# B&R Automation Studio project Task_2
Automation Studio 4.9

## Logical view

Binary libraries used (declarations not repeated): operator, runtime, astime, AsIecCon, Acp10man, Acp10par, NcGlobal, Acp10_MC, sys_lib, brsystem, Acp10sim, MpAxis, MpCom, MpBase, AsTCP, standard, AsArLog, AsBrStr

### Global.var - Global variables
```iecst
VAR
	EmergencyLight : BOOL;
END_VAR
VAR RETAIN
	MyGlobal : {REDUND_UNREPLICABLE} UDINT := 10;
END_VAR
VAR
	CUTTER_END_POSE : REAL := 50.0;
END_VAR
VAR CONSTANT
	BELT_DISTANCE : REAL := 100.0;
	CUTTER_SPEED : REAL := 100.0;
END_VAR
VAR
	RealConveyorSpeed : INT;
	CONVEYOR_SPEED : {REDUND_UNREPLICABLE} INT := 1000;
	gAxis01 : ACP10AXIS_typ;
	gAxis02 : ACP10AXIS_typ;
	START_BUTTON : BOOL;
	TRIGGER_INPUT : BOOL;
	EMERGENCY_STOP : BOOL;
	GreenLight : BOOL;
	RedLight : BOOL;
	CutterPosition : LREAL;
	ConveyorPosition : LREAL;
	STOP : BOOL;
	ERROR_RESET : BOOL;
END_VAR
```

### Package Logical/Libraries - Global libraries

### MNG_Global.hpp
```cpp
#ifndef  _MNGGLOBAL_HPP_
#define _MNGGLOBAL_HPP_

#include <mng_globalTYP.h>

    typedef struct {

		signed short NumSignals;

        /* BOOL Emergency_Button_ButtonToggle */
        BOOL Emergency_Button_ButtonToggle;
        /* BOOL Yellow_Button_ButtonPress */
        BOOL Yellow_Button_ButtonPress;
        /* BOOL White_Button_ButtonPress */
        BOOL White_Button_ButtonPress;
        /* BOOL Start_Button_ButtonPress */
        BOOL Start_Button_ButtonPress;
        /* BOOL Stop_Button_ButtonPress */
        BOOL Stop_Button_ButtonPress;
        /* REAL Knob_0_AXIS */
        REAL Knob_0_AXIS;
        /* REAL Knob_1_AXIS */
        REAL Knob_1_AXIS;
        /* REAL Knob_2_AXIS */
        REAL Knob_2_AXIS;
        /* REAL Knob_3_AXIS */
        REAL Knob_3_AXIS;
        /* REAL Shaft_1_AXIS */
        REAL Shaft_1_AXIS;
        /* BOOL Shaft_1_LBK */
        BOOL Shaft_1_LBK;
        /* BOOL Shaft_1_LFR */
        BOOL Shaft_1_LFR;
        /* REAL Shaft_0_AXIS */
        REAL Shaft_0_AXIS;
        /* BOOL Shaft_0_LBK */
        BOOL Shaft_0_LBK;
        /* BOOL Shaft_0_LFR */
        BOOL Shaft_0_LFR;

        } ComTCP_INPUTS_32BIT_FWRD;

    typedef struct {

		signed short NumSignals;

        /* UDINT Yellow_light_Key */
        UDINT Yellow_light_Key;
        /* UDINT Stop_light_Key */
        UDINT Stop_light_Key;
        /* UDINT White_light_Key */
        UDINT White_light_Key;
        /* UDINT Green_light_Key */
        UDINT Green_light_Key;
        /* REAL Shaft_0_ACT_POS */
        REAL Shaft_0_ACT_POS;
        /* REAL Shaft_1_ACT_POS */
        REAL Shaft_1_ACT_POS;

        } ComTCP_OUTPUTS_32BIT_FWRD;

#endif
```

### Library Logical/Libraries/CAMlib (IEC)

#### Types.typ - Exported data types
```iecst
TYPE
	GA_State :
		(
		NotPowered,
		WaitEnable,
		WaitPower,
		Powered,
		CheckCommand,
		MoveVelocity,
		CheckVelocity,
		MoveAdditive,
		CheckAdditiveUpdate,
		AxisHalt,
		AxisStop,
		CheckCamUpdate,
		CheckCam,
		MoveCam,
		CheckVelocityUpdate,
		AxisEmergency
		);
	COMMANDS :
		(
		NONE,
		MOVE_VELOCITY,
		MOVE_ADDITIVE,
		AXIS_HALT,
		AXIS_STOP,
		MOVE_CAM,
		AXIS_EMERGENCY
		);
END_TYPE
```

#### CAMlib.fun - Exported functions and function blocks
```iecst
{REDUND_ERROR} FUNCTION_BLOCK CamFB (*TODO: Add your comment here*) (*$GROUP=User,$CAT=User,$GROUPICON=User.png,$CATICON=User.png*)
	VAR_INPUT
		AxisOperation : INT;
		AxisCommand : COMMANDS;
		Axis : UDINT;
		MpLinkMaster : UDINT;
		MpLink : UDINT;
		Slave : UDINT;
		CamTable : ARRAY[0..4] OF STRING[12];
		Position : REAL;
		Velocity : REAL;
		Acceleration : REAL;
		Deceleration : REAL;
		Jerk : REAL;
		Direction : USINT;
		ArraySize : INT;
		Scale : REAL;
		Offset : REAL;
		RatioNumerator : INT;
		CamID : USINT;
		CamActivated : BOOL;
		RatioDenominator : INT;
		CouplingParam : MpAxisCouplingParType;
		Param : MpAxisBasicParType;
	END_VAR
	VAR_OUTPUT
		CommandExecuted : BOOL;
		CommandAborted : BOOL;
		Error : BOOL;
		ErrorID : UINT;
		AxisErrorID : UINT;
		AxisErrorCount : UINT;
		AxisNotInitialized : BOOL;
		Status : WORD;
		ActualVelocity : REAL;
		ActualPosition : LREAL;
	END_VAR
	VAR_IN_OUT
		AxisEnable : BOOL;
	END_VAR
	VAR
		MpAxisCoupling : MpAxisCoupling;
		MpAxisBasic : MpAxisBasic;
		OldVelocity : REAL;
		AxisState : GA_State;
		OldCamID : USINT;
	END_VAR
END_FUNCTION_BLOCK
```

#### CamFB.st
```iecst
(* TODO: Add your comment here *)
FUNCTION_BLOCK CamFB

	CASE (AxisState) OF
		NotPowered:
			IF AxisEnable THEN
				MpAxisBasic.Enable := TRUE;
				AxisState := WaitEnable;
			END_IF;

		WaitEnable:
			IF MpAxisBasic.Active THEN
				MpAxisBasic.Power := TRUE;
				AxisState := WaitPower; //ready state in the prof's slides
			END_IF;

		WaitPower:
			IF  MpAxisBasic.PowerOn THEN
				MpAxisBasic.Home := TRUE;
				AxisState := Powered;
			END_IF;

		Powered:
			IF MpAxisBasic.IsHomed THEN // condition for the homing
				MpAxisBasic.Home := FALSE;
				AxisEnable := FALSE;
				CommandExecuted := TRUE;
				MpAxisCoupling.Enable := TRUE;
				AxisState := CheckCommand; //ready state in the prof's slides
			END_IF;

		CheckCommand:
			IF AxisCommand = MOVE_VELOCITY THEN
				CommandExecuted := FALSE;
				MpAxisBasic.MoveAdditive := FALSE;
				MpAxisBasic.Update := TRUE;
				// MpAxisBasic.MoveVelocity := TRUE;  // <------ Come se ricevesse velocità nulla
				AxisState := CheckVelocityUpdate;
			END_IF;

			IF AxisCommand = MOVE_ADDITIVE THEN
				CommandExecuted := FALSE;
				MpAxisBasic.MoveVelocity := FALSE;
				MpAxisBasic.MoveAdditive := TRUE;
				MpAxisBasic.Update := TRUE;
				AxisState := CheckAdditiveUpdate; //CheckAdditiveUpdate;
			END_IF;

			IF AxisCommand = AXIS_STOP THEN
				CommandExecuted := FALSE;
				MpAxisBasic.MoveVelocity := FALSE;
				MpAxisBasic.MoveAdditive := FALSE;
				MpAxisBasic.Stop := TRUE;
				AxisState := AxisStop;
			END_IF;

			IF AxisCommand = AXIS_EMERGENCY THEN
				CommandExecuted := FALSE;
				MpAxisBasic.MoveVelocity := FALSE;
				MpAxisBasic.MoveAdditive := FALSE;
				MpAxisBasic.Stop := TRUE;
				AxisState := AxisEmergency;
			END_IF;

			IF AxisCommand = MOVE_CAM AND CamActivated THEN
				CommandExecuted := FALSE;
				MpAxisCoupling.Cam := TRUE;
				AxisState := MoveCam;
			END_IF;

	(*IF AxisCommand = NONE THEN
		CommandExecuted := FALSE;
	END_IF*)

// command states
		MoveVelocity:
			IF MpAxisBasic.InVelocity THEN  // <------- Siccome la velocità è nulls lo esegue subito
				CommandExecuted := TRUE;
				AxisState := CheckVelocity;
			END_IF;

			IF (AxisCommand <> MOVE_VELOCITY) THEN
				CommandExecuted := FALSE;
				MpAxisBasic.MoveVelocity := FALSE;
				AxisState := CheckCommand;
			END_IF;

		CheckVelocity:
			IF (Param.Velocity <> OldVelocity) THEN
				OldVelocity := Param.Velocity;
				MpAxisBasic.Update := TRUE;
				AxisState := CheckVelocityUpdate;
			END_IF;
			IF (AxisCommand <> MOVE_VELOCITY) THEN
				CommandExecuted := FALSE;
				MpAxisBasic.MoveVelocity := FALSE;
				AxisState := CheckCommand;
			END_IF;

		CheckVelocityUpdate:
			IF MpAxisBasic.UpdateDone THEN
				MpAxisBasic.Update := FALSE;
				MpAxisBasic.MoveVelocity := TRUE;
				CommandExecuted := FALSE;
				AxisState := MoveVelocity;
			END_IF;

		MoveAdditive:
			IF MpAxisBasic.InPosition THEN
				MpAxisBasic.MoveAdditive := FALSE;
				AxisCommand := NONE;
				AxisState := CheckCommand;
				CommandExecuted := TRUE;
			ELSIF (AxisCommand <> MOVE_ADDITIVE) THEN
				MpAxisBasic.MoveAdditive := FALSE;
				CommandExecuted := FALSE;
				AxisState := CheckCommand;
			END_IF;

		CheckAdditiveUpdate:
			IF MpAxisBasic.UpdateDone THEN
				MpAxisBasic.Update := FALSE;
				MpAxisBasic.MoveAdditive := TRUE;
				CommandExecuted := FALSE;
					AxisState := MoveAdditive;
			END_IF;

		AxisStop:
			IF MpAxisBasic.Stopped THEN
				CommandExecuted := TRUE;
				MpAxisBasic.Stop := FALSE;
				MpAxisBasic.Power := FALSE; // The power is disabled for the same reason
				// MpAxisBasic.Enable := FALSE;
				// MpAxisCoupling.Enable := FALSE;
				MpAxisCoupling.Cam := FALSE;
				AxisCommand := NONE;
				AxisState := NotPowered; // It goes to the NotPowered state to perform a full reset of the system
			END_IF;

		AxisEmergency:
			IF MpAxisBasic.Stopped THEN
				CommandExecuted := TRUE;
				MpAxisBasic.Stop := FALSE;
				MpAxisBasic.Power := FALSE; // The power is disabled for the same reason
				// MpAxisBasic.Enable := FALSE;
				// MpAxisCoupling.Enable := FALSE;
				MpAxisCoupling.Cam := FALSE;
				AxisCommand := NONE;
				AxisState := NotPowered; // It goes to the NotPowered state to perform a full reset of the system
			END_IF;

			// memo, we don't check the mpaxiscoupling.active -> WARNING

		MoveCam:
			IF MpAxisCoupling.InSync THEN
				CommandExecuted := TRUE;
				AxisState := CheckCam;
			END_IF
			IF (AxisCommand <> MOVE_CAM) THEN
				CommandExecuted := FALSE;
				MpAxisCoupling.Cam := FALSE;
				MpAxisCoupling.Enable := FALSE;
				AxisState := CheckCommand;
			END_IF;
		CheckCam:
			IF CamID <> OldCamID THEN
				OldCamID := CamID;
				CommandExecuted := FALSE;
				MpAxisCoupling.Update := TRUE;
				AxisState := CheckCamUpdate;
			END_IF
			IF (AxisCommand <> MOVE_CAM) THEN
				CommandExecuted := FALSE;
				MpAxisCoupling.Cam := FALSE;
				MpAxisCoupling.Enable := FALSE;
				AxisState := CheckCommand;
			END_IF;

		CheckCamUpdate:
			IF MpAxisCoupling.UpdateDone THEN
				MpAxisCoupling.Update := FALSE;
				AxisState := MoveCam;
			END_IF;

	END_CASE

	MpAxisBasic.Axis := Axis;
	MpAxisBasic.MpLink := MpLink;

	MpAxisBasic.Parameters	:= ADR(Param);
	ActualPosition := MpAxisBasic.Position;

	MpAxisBasic();

	IF CamActivated THEN
		MpAxisCoupling.MpLinkMaster	:= MpLinkMaster;
		MpAxisCoupling.MpLink := MpLink;
		CouplingParam.Cam.CamTableID := CamID;
		CouplingParam.Cam.CamTable := CamTable;
		MpAxisCoupling.Parameters := ADR(CouplingParam);
		MpAxisCoupling();
	END_IF

END_FUNCTION_BLOCK
```

### Package Logical/gAxis02obj - gAxis02obj

### gAxis02i.ax
```
InitParameter (Version=5.24.1, NcSwId=Acp10)
  ACP10AXIS_typ:
    dig_in:
      level:
        reference = ncACTIV_HI
        pos_hw_end = ncACTIV_HI
        neg_hw_end = ncACTIV_HI
        trigger1 = ncACTIV_HI
        trigger2 = ncACTIV_HI
    encoder_if:
      parameter:
        count_dir = ncSTANDARD
        scaling:
          load:
            units = 360
            rev_motor = 1
    limit:
      parameter:
        v_pos = 10000
        v_neg = 10000
        a1_pos = 50000
        a2_pos = 50000
        a1_neg = 50000
        a2_neg = 50000
        t_jolt = 0
        t_in_pos = 0
        pos_sw_end = 2000000000
        neg_sw_end = -2000000000
        ds_warning = 500
        ds_stop = 1000
        a_stop = 1.0e30
        dv_stop = 0
        dv_stop_mode = ncOFF
    controller:
      mode = ncPOSITION
      position:
        kv = 349.0
        tn = 0
        t_predict = 0.0004
        t_total = 0.0004
        p_max = 1.0e30
        i_max = 0
      speed:
        kv = 0.65
        tn = 0
        t_filter = 0.0
        isq_filter1:
          type = ncOFF
          a0 = 0.0
          a1 = 0.0
          b0 = 0.0
          b1 = 0.0
          b2 = 0.0
          c0_par_id = 0
          c1_par_id = 0
        isq_filter2:
          type = ncOFF
          a0 = 0.0
          a1 = 0.0
          b0 = 0.0
          b1 = 0.0
          b2 = 0.0
          c0_par_id = 0
          c1_par_id = 0
        isq_filter3:
          type = ncOFF
          a0 = 0.0
          a1 = 0.0
          b0 = 0.0
          b1 = 0.0
          b2 = 0.0
          c0_par_id = 0
          c1_par_id = 0
      uf:
        type = ncLINEAR + ncCORRECTION
        auto_config = ncMOTOR_PAR
        u0 = 0
        un = 0
        fn = 50.0
        k_f_slip = 0
      ff:
        mode = ncSTANDARD
        torque_load = 0.0
        torque_pos = 0.0
        torque_neg = 0.0
        kv_torque = 0.0
        inertia = 0.0
        t_filter_a = 0.0
      fb:
        mode = ncSTANDARD
        speed_mix_ratio = 0.0
        speed_kv = 2.0
      model:
        mass1:
          inertia = 0
          viscous_friction = 0
        mass2:
          inertia = 0
          viscous_friction = 0
          stiffness = 0
          damping = 0
    move:
      stop:
        parameter[0]:
          decel_ramp = ncA_LIMIT
          controller = ncON
        parameter[1]:
          decel_ramp = ncA_LIMIT
          controller = ncON
        parameter[2]:
          decel_ramp = ncA_LIMIT
          controller = ncON
        parameter[3]:
          decel_ramp = ncA_LIMIT
          controller = ncON
        quickstop:
          decel_ramp = ncA_LIMIT
          t_jolt = 0
        drive_error:
          decel_ramp = ncA_LIMIT
      homing:
        parameter:
          s = 0
          v_switch = 5000
          v_trigger = 500
          a = 50000
          mode = ncDIRECT
          edge_sw = ncPOSITIVE
          start_dir = ncPOSITIVE
          trigg_dir = ncPOSITIVE
          ref_pulse = ncOFF
          fix_dir = ncOFF
          tr_s_block = 0
          torque_lim = 0
          ds_block = 0
          ds_stop = 0
      basis:
        parameter:
          v_pos = 5000
          v_neg = 5000
          a1_pos = 50000
          a2_pos = 50000
          a1_neg = 50000
          a2_neg = 50000
    message:
      text:
        parameter:
          format = ncBREAK
          columns = 80
          data_modul = acp10etxen
```

### Program Logical/PROGRAM1 (IEC)

#### Types.typ
```iecst
TYPE
	State_type :
		(
		CutterMoveBackward,
		CutterCompleted,
		CutterMoveForward,
		ConveyorStopping,
		ConveyorMoving,
		ConveyorStarting,
		AxisEnabled,
		InitializeAxis,
		CutterBackward,
		CutterForward,
		ConveyorHolding,
		WaitProduct,
		Initialize,
		Init,
		StopState,
		HaltState,
		WaitForConveyor,
		CheckReset
		);
END_TYPE
```

#### Variables.var
```iecst
VAR
	Address : UDINT;
	MachineState : State_type;
	ConveyorEnable : BOOL;
	CutterEnable : BOOL;
	Cutter : CamFB;
	Conveyor : CamFB;
	InitializeConveyor : BOOL;
	InitializeCutter : BOOL;
	ConveyorDisable : BOOL;
	CutterDisable : BOOL;
	ConveyorState : State_type;
	CutterState : State_type;
	ConveyorAxisEnable : BOOL;
	CutterAxisEnable : BOOL;
	FutureStop : BOOL;
	CoveyorState : BOOL;
	ConveyorStopped : BOOL;
	CutterStopped : BOOL;
	ConveyorParameters : MpAxisBasicParType;
	CutterParameters : MpAxisBasicParType;
	EmergencyStateMachine : INT;
	ToggleLights : BOOL;
	Count : DINT;
END_VAR
```

#### Main.st
```iecst
PROGRAM _INIT
	(* Insert code here *)
	MachineState := Init;
	ConveyorState := Init;
	CutterState := Init;

END_PROGRAM

PROGRAM _CYCLIC

	// STOP indicates an emergency stop, it is not a stop in normal conditions
	CASE EmergencyStateMachine OF
		0 :
			IF EMERGENCY_STOP THEN
				MachineState := StopState;
				ConveyorState := StopState;
				CutterState := StopState;
				Conveyor.AxisCommand := AXIS_STOP;
				Cutter.AxisCommand := AXIS_STOP;
				EmergencyStateMachine := 1;
			END_IF
		1 :
			IF NOT EMERGENCY_STOP AND CutterStopped AND ConveyorStopped THEN
				EmergencyStateMachine := 0;
			END_IF
	END_CASE

	IF STOP THEN
		FutureStop := TRUE;
	END_IF

	// GLOBAL STATE MACHINE
	CASE MachineState OF
		Init: // Initial configuration state
			IF START_BUTTON THEN
				InitializeConveyor := TRUE;
				InitializeCutter := TRUE;
				MachineState := Initialize;
			END_IF
		Initialize: // initialization - Power and Homing (This operations are implemented inside the function block)
			IF NOT InitializeConveyor AND NOT InitializeCutter THEN
				ConveyorEnable := TRUE;
				MachineState := WaitProduct;
			END_IF
		WaitProduct: // It waits for a trigger
			IF NOT ConveyorEnable AND TRIGGER_INPUT THEN
				ConveyorDisable := TRUE;
				MachineState := ConveyorHolding;
			END_IF
			// STOP
			IF FutureStop THEN
				MachineState := HaltState;
			END_IF

		ConveyorHolding: // Stop the Conveyor
			IF NOT ConveyorDisable THEN
				CutterEnable := TRUE;
				MachineState := CutterForward;
			END_IF
		CutterForward: // Cut
			IF NOT CutterEnable THEN
				CutterDisable := TRUE;
				MachineState := CutterBackward;
			END_IF
		CutterBackward: // Go back
			IF NOT CutterDisable THEN
				ConveyorEnable := TRUE;
				MachineState := WaitProduct;
			END_IF

		// Emergency stop
		StopState:
			IF NOT EMERGENCY_STOP AND ConveyorStopped AND CutterStopped THEN
				MachineState := CheckReset;
			END_IF
		CheckReset:
			IF ERROR_RESET THEN
				MachineState := Init;
				ConveyorStopped := FALSE;
				CutterStopped := FALSE;
				FutureStop := FALSE;
			END_IF
			// CAN BE ERASED
		// CAN BE ERASED
		HaltState:
			IF ConveyorStopped AND CutterStopped THEN
				MachineState := Init;
				ConveyorStopped := FALSE;
				CutterStopped := FALSE;
				FutureStop := FALSE;
			END_IF

	END_CASE

	// CONVEYOR STATE MACHINE
	CASE ConveyorState OF
		Init:
			IF InitializeConveyor THEN
				ConveyorAxisEnable := TRUE;
				ConveyorState := InitializeAxis;
			END_IF
		InitializeAxis:
			IF NOT ConveyorAxisEnable THEN
				InitializeConveyor := FALSE;
				ConveyorState := AxisEnabled;
			END_IF
		AxisEnabled:
			IF ConveyorEnable AND NOT FutureStop THEN
				Conveyor.AxisCommand := MOVE_VELOCITY;
				ConveyorState := ConveyorStarting;
			ELSIF FutureStop THEN
				Conveyor.AxisCommand := AXIS_STOP;
				ConveyorState := HaltState;
			END_IF
		ConveyorStarting:
			IF Conveyor.CommandExecuted THEN
				ConveyorEnable := FALSE;
				ConveyorState := ConveyorMoving;
			END_IF
		ConveyorMoving:
			IF ConveyorDisable AND NOT FutureStop THEN
				Conveyor.AxisCommand := MOVE_ADDITIVE;
				ConveyorState := ConveyorStopping;
			ELSIF FutureStop THEN
				Conveyor.AxisCommand := AXIS_STOP;
				ConveyorState := HaltState;
			END_IF
		ConveyorStopping:
			IF Conveyor.CommandExecuted THEN
				ConveyorDisable := FALSE;
				ConveyorState := AxisEnabled;
			END_IF

		// EMERGENCY STOP
		StopState:
			IF NOT EMERGENCY_STOP AND Conveyor.CommandExecuted THEN
				ConveyorEnable := FALSE;
				ConveyorDisable := FALSE;
				ConveyorStopped := TRUE;
				ConveyorState := Init;
			END_IF

		HaltState:
			IF Conveyor.CommandExecuted THEN
				ConveyorDisable := FALSE;
				ConveyorEnable := FALSE;
				ConveyorStopped := TRUE;
				ConveyorState := Init;
			END_IF
	END_CASE

	// CUTTER STATE MACHINE
	CASE CutterState OF
		Init:
			IF InitializeCutter THEN
				CutterAxisEnable := TRUE;
				CutterState := InitializeAxis;
			END_IF
		InitializeAxis:
			IF NOT CutterAxisEnable THEN
				InitializeCutter := FALSE;
				CutterState := AxisEnabled;
			END_IF
		AxisEnabled:
			IF ConveyorDisable AND NOT FutureStop THEN
				CutterState := WaitForConveyor;
			ELSIF FutureStop THEN
				Cutter.AxisCommand := AXIS_STOP;
				CutterState := HaltState;
			END_IF
		WaitForConveyor:
			IF CutterEnable THEN
				Cutter.Param.Distance := CUTTER_END_POSE; // Added by me
				Cutter.AxisCommand := MOVE_ADDITIVE;
				CutterState := CutterMoveForward;
			END_IF
		CutterMoveForward:
			IF Cutter.CommandExecuted THEN
				CutterEnable := FALSE;
				CutterState := CutterCompleted;
			END_IF
		CutterCompleted:
			IF CutterDisable THEN
				Cutter.Param.Distance := -CUTTER_END_POSE; // Added by me
				Cutter.AxisCommand := MOVE_ADDITIVE;
				CutterState := CutterMoveBackward;
			END_IF
		CutterMoveBackward:
			IF Cutter.CommandExecuted THEN
				CutterDisable := FALSE;
				CutterState := AxisEnabled;
			END_IF

		// EMERGENCY STOP
		StopState:
			IF NOT EMERGENCY_STOP AND Cutter.CommandExecuted THEN
				CutterEnable := FALSE;
				CutterDisable := FALSE;
				CutterStopped := TRUE;
				CutterState := Init;
			END_IF

		HaltState:
			IF Cutter.CommandExecuted THEN
				CutterDisable := FALSE;
				CutterEnable := FALSE;
				CutterStopped := TRUE;
				CutterState := Init;
			END_IF
	END_CASE

	// Counter for blink
	Count := Count + 1;
	IF Count = 10 THEN
		ToggleLights := TRUE;
		Count := 0;
	ELSE
		ToggleLights := FALSE;
	END_IF

	// LIGHTS
	IF MachineState = Init THEN
		IF ToggleLights THEN
			GreenLight := NOT GreenLight;
		END_IF
		RedLight := FALSE;
		EmergencyLight := FALSE;

	ELSIF MachineState <> HaltState AND MachineState <> StopState AND MachineState <> CheckReset THEN
		GreenLight := TRUE;
		RedLight := TRUE;
		EmergencyLight := FALSE;
	ELSIF MachineState = StopState OR MachineState = CheckReset THEN
		GreenLight := FALSE;
		RedLight := FALSE;
		IF ToggleLights THEN
			EmergencyLight := NOT EmergencyLight;
		END_IF
	END_IF

	Conveyor.Axis := ADR(gAxis01);
	Conveyor.MpLink := ADR(gAxisConveyor);
	//Conveyor.Param := ConveyorParameters; //  <------ non vengono passati bene

	Conveyor.Param.Distance := 2*BELT_DISTANCE;
	RealConveyorSpeed := CONVEYOR_SPEED/10;
	Conveyor.Param.Velocity := INT_TO_REAL(RealConveyorSpeed);
	Conveyor.Param.Acceleration := 50;
	Conveyor.Param.Deceleration := 50;

	Conveyor(AxisEnable := ConveyorAxisEnable);
	ConveyorPosition := Conveyor.ActualPosition;

	Cutter.Axis := ADR(gAxis02);
	Cutter.MpLink := ADR(gAxisCutter);
	//Cutter.Param := CutterParameters; //  <------ non vengono passati bene

	Cutter.Param.Velocity := CUTTER_SPEED;
	Cutter.Param.Acceleration := 50;
	Cutter.Param.Deceleration := 50;

	Cutter(AxisEnable := CutterAxisEnable);
	CutterPosition := Cutter.ActualPosition;

END_PROGRAM

PROGRAM _EXIT
	(* Insert code here *)

END_PROGRAM
```

### MNG_Package.typ
```iecst
(*                                                                            *)
(* File generated by the B&R AS 4 control config generator                    *)
(*                                                                            *)
(*     Provider: machineering                                                 *)
(*  Application: industrialPhysics_2.4.master                                 *)
(* Architecture: Windows 64 Bit                                               *)
(*      Version: 2.4.10491.master                                             *)
(*        Build: 164f85bec                                                    *)
(*         Date: 2020-03-30, Time: 13:49:25                                   *)
(*                                                                            *)

TYPE
ComTCP_INPUTS_32BIT : STRUCT

		NumSignals	: INT := 15;

        Emergency_Button_ButtonToggle : BOOL := 0;
        (* BOOL Emergency_Button_ButtonToggle *)
        Yellow_Button_ButtonPress : BOOL := 0;
        (* BOOL Yellow_Button_ButtonPress *)
        White_Button_ButtonPress : BOOL := 0;
        (* BOOL White_Button_ButtonPress *)
        Start_Button_ButtonPress : BOOL := 0;
        (* BOOL Start_Button_ButtonPress *)
        Stop_Button_ButtonPress : BOOL := 0;
        (* BOOL Stop_Button_ButtonPress *)
        Knob_0_AXIS : REAL := 0.0;
        (* REAL Knob_0_AXIS *)
        Knob_1_AXIS : REAL := 0.0;
        (* REAL Knob_1_AXIS *)
        Knob_2_AXIS : REAL := 0.0;
        (* REAL Knob_2_AXIS *)
        Knob_3_AXIS : REAL := 0.0;
        (* REAL Knob_3_AXIS *)
        Shaft_1_AXIS : REAL := 0.0;
        (* REAL Shaft_1_AXIS *)
        Shaft_1_LBK : BOOL := 0;
        (* BOOL Shaft_1_LBK *)
        Shaft_1_LFR : BOOL := 0;
        (* BOOL Shaft_1_LFR *)
        Shaft_0_AXIS : REAL := 0.0;
        (* REAL Shaft_0_AXIS *)
        Shaft_0_LBK : BOOL := 0;
        (* BOOL Shaft_0_LBK *)
        Shaft_0_LFR : BOOL := 0;
        (* BOOL Shaft_0_LFR *)

	END_STRUCT;

ComTCP_OUTPUTS_32BIT : STRUCT

		NumSignals	: INT := 6;

        Yellow_light_Key : UDINT := 0;
        (* UDINT Yellow_light_Key *)
        Stop_light_Key : UDINT := 0;
        (* UDINT Stop_light_Key *)
        White_light_Key : UDINT := 0;
        (* UDINT White_light_Key *)
        Green_light_Key : UDINT := 0;
        (* UDINT Green_light_Key *)
        Shaft_0_ACT_POS : REAL := 0.0;
        (* REAL Shaft_0_ACT_POS *)
        Shaft_1_ACT_POS : REAL := 0.0;
        (* REAL Shaft_1_ACT_POS *)

	END_STRUCT;

END_TYPE
```

### MNG_Package.var
```iecst
(*                                                                            *)
(* File generated by the B&R AS 4 control config generator                    *)
(*                                                                            *)
(*     Provider: machineering                                                 *)
(*  Application: industrialPhysics_2.4.master                                 *)
(* Architecture: Windows 64 Bit                                               *)
(*      Version: 2.4.10491.master                                             *)
(*        Build: 164f85bec                                                    *)
(*         Date: 2020-03-30, Time: 13:49:25                                   *)
(*                                                                            *)
VAR
	ComTCP_SimInputs : ComTCP_INPUTS_32BIT := (0);
	ComTCP_SimOutputs : ComTCP_OUTPUTS_32BIT := (0);
	ComTCP_SimServerAddress : STRING[15] := '127.0.0.1';
	ComTCP_SimServerPort : UINT := 5000;
	ComTCP_SimSendCycleTime : TIME := T#10ms;
	ComTCP_SimActive : BOOL := FALSE;
	ResetButton : BOOL;
END_VAR
```

### Program Logical/OutputBridge (IEC)

#### Main.st
```iecst
PROGRAM _INIT
	(* Insert code here *)

END_PROGRAM

PROGRAM _CYCLIC
	(* Insert code here *)
	ComTCP_SimOutputs.Green_light_Key := GreenLight;
	ComTCP_SimOutputs.Stop_light_Key := RedLight;
	ComTCP_SimOutputs.Yellow_light_Key := EmergencyLight;
	ComTCP_SimOutputs.Shaft_0_ACT_POS := LREAL_TO_REAL(ConveyorPosition);
	ComTCP_SimOutputs.Shaft_1_ACT_POS := LREAL_TO_REAL(CutterPosition);

END_PROGRAM

PROGRAM _EXIT
	(* Insert code here *)

END_PROGRAM
```

### Program Logical/MC_mmg (IEC)

#### Main.st - Init, cyclic, exit code
```iecst
PROGRAM _INIT
	// executed only once at the start

	Cutter.CamActivated := TRUE;

	Cutter.CamTable[0]	:= 'standstill';		// since we have only 1 cam we fill the first array,
	Cutter.CamTable[1]	:= 'Cam';
	Cutter.CamID := 0;					// the default value is 0
	CouplingParameters.RatioDenominator := 1;

	// CouplingParameters.Cam.CamTable[1]	:= 'Cam1';		// it's the name of the cam folder and the number of the cam

	// in the mpaxiscoupling_cutter --> info section --> we can see if master and slave can be synchronized
	// either master and slave start to false, in order to have the MasterReady = TRUE the conveyor must be homed
	// so the IsHomed flag goes to TRUE then the MasterReady = TRUE
	// the MasterReady = TRUE when Conveyor is Homed, but since I want to move it I need to set Power = TRUE (NOTE: In order to have MasterReady = TRUE, Power = TRUE is not necessary)
	// The SlaveReady = TRUE when the Cutter is Homed and Powered (Power = TRUE).
	// setting the CAM = TRUE in the cutter PLCOpen = Sync
	// in coupling parameters it's possible to choose the numerator for the slave and the denominator for the slave, at the moment with a RatioNumerator = 360
	// the slave does a complete rotation represents the cut task
	// RatioNumerator and RatioDenominator are the stretching factor of the normalized cam    (180 means 180° of range)

	(* Insert code here *)
	MachineState := Init;
	ConveyorState := Init;
	CutterState := Init;

END_PROGRAM

PROGRAM _CYCLIC

	// STOP indicates an emergency stop, it is not a stop in normal conditions
	CASE EmergencyStateMachine OF
		0 :
			IF EMERGENCY_STOP THEN
				MachineState := StopState;
				ConveyorState := StopState;
				CutterState := StopState;
				Conveyor.AxisCommand := AXIS_EMERGENCY;
				Cutter.AxisCommand := AXIS_EMERGENCY;
				EmergencyStateMachine := 1;
			END_IF
		1 :
			IF NOT EMERGENCY_STOP AND CutterStopped AND ConveyorStopped THEN
				EmergencyStateMachine := 0;
			END_IF
	END_CASE

	(*IF EMERGENCY_STOP AND THEN
		MachineState := StopState;
		ConveyorState := StopState;
		CutterState := StopState;
		Conveyor.AxisCommand := AXIS_HALT;
		Cutter.AxisCommand := AXIS_HALT;
	END_IF*)

	IF STOP THEN
		FutureStop := TRUE;
	END_IF

	// GLOBAL STATE MACHINE
	CASE MachineState OF
		Init: // Initial configuration state
			IF START_BUTTON THEN
				InitializeConveyor := TRUE;
				InitializeCutter := TRUE;
				MachineState := Initialize;
			END_IF
		Initialize: // initialization - Power and Homing (This operations are implemented inside the function block)
			IF NOT InitializeConveyor AND NOT InitializeCutter THEN
				ConveyorEnable := TRUE;
				MachineState := WaitProduct;
			END_IF
		WaitProduct: // It waits for a trigger
			IF NOT ConveyorEnable AND TRIGGER_INPUT THEN
				CutterEnable := TRUE;
				MachineState := CutterForward;
			END_IF
			// STOP
			IF FutureStop AND CutterPosition = 0.0 THEN
				MachineState := HaltState;
			END_IF
		CutterForward: // Cut
			IF NOT CutterEnable THEN
				CutterDisable := TRUE;
				MachineState := CutterBackward;
			END_IF
		CutterBackward: // Go back
			IF NOT CutterDisable THEN
				// ConveyorEnable := TRUE;
				MachineState := WaitProduct;
			END_IF

			// Emergency stop
		StopState:
			IF NOT EMERGENCY_STOP AND ConveyorStopped AND CutterStopped THEN
				MachineState := CheckReset;
			END_IF
		CheckReset:
			IF ERROR_RESET THEN
				MachineState := Init;
				ConveyorStopped := FALSE;
				CutterStopped := FALSE;
				FutureStop := FALSE;
			END_IF
			// CAN BE ERASED
		HaltState:
			IF ConveyorStopped AND CutterStopped THEN
				MachineState := Init;
				ConveyorStopped := FALSE;
				CutterStopped := FALSE;
				FutureStop := FALSE;
			END_IF

	END_CASE

	// CONVEYOR STATE MACHINE
	CASE ConveyorState OF
		Init:
			IF InitializeConveyor THEN
				ConveyorAxisEnable := TRUE;
				ConveyorState := InitializeAxis;
			END_IF
		InitializeAxis:
			IF NOT ConveyorAxisEnable THEN
				InitializeConveyor := FALSE;
				ConveyorState := AxisEnabled;
			END_IF
		AxisEnabled:
			IF ConveyorEnable AND (NOT FutureStop OR CutterPosition <> 0.0) THEN
				Conveyor.AxisCommand := MOVE_VELOCITY;
				ConveyorState := ConveyorStarting;
			ELSIF FutureStop AND CutterPosition = 0.0 THEN
				Conveyor.AxisCommand := AXIS_STOP;
				ConveyorState := HaltState;
			END_IF
		ConveyorStarting:
			IF Conveyor.CommandExecuted THEN
				ConveyorEnable := FALSE;
				ConveyorState := ConveyorMoving;
			END_IF
		ConveyorMoving:
			IF FutureStop AND NOT CutterWorking THEN
				Conveyor.AxisCommand := AXIS_STOP;
				ConveyorState := HaltState;
			END_IF

			// EMERGENCY STOP
		StopState:
			IF NOT EMERGENCY_STOP AND Conveyor.CommandExecuted THEN
				ConveyorEnable := FALSE;
				ConveyorDisable := FALSE;
				ConveyorStopped := TRUE;
				ConveyorState := Init;
			END_IF

		HaltState:
			IF Conveyor.CommandExecuted THEN
				ConveyorDisable := FALSE;
				ConveyorEnable := FALSE;
				ConveyorStopped := TRUE;
				ConveyorAxisEnable := FALSE;
				ConveyorState := Init;
			END_IF
	END_CASE

	// CUTTER STATE MACHINE
	CASE CutterState OF
		Init:
			IF InitializeCutter THEN
				CutterAxisEnable := TRUE;
				CutterState := InitializeAxis;
			END_IF
		InitializeAxis:
			IF NOT CutterAxisEnable THEN
				Cutter.AxisCommand := MOVE_CAM;
				CutterState := CamEnabled;
			END_IF
		CamEnabled:
			IF Conveyor.CommandExecuted THEN
				InitializeCutter := FALSE;
				CutterState := AxisEnabled;
			END_IF
		AxisEnabled:
			IF CutterEnable AND NOT FutureStop THEN
				CutterWorking := TRUE;
				Cutter.CamID := 1;
				CutterState := CheckCamUpdate1;
			ELSIF FutureStop THEN
				Cutter.AxisCommand := AXIS_STOP;
				CutterState := HaltState;
			END_IF

		CheckCamUpdate1:
			IF Cutter.CommandExecuted THEN
				// cambio camma
				CutterEnable := FALSE;
				CutterState := CutterMoveForward;
			END_IF
		CutterMoveForward:
			IF CutterPosition <> 0.0 THEN
				// cambio camma
				Cutter.CamID := 0;
				CutterState := CheckCamUpdate2;
			END_IF
		CheckCamUpdate2:
			IF Cutter.CommandExecuted THEN
				// cambio camma
				CutterState := CutterCompleted;
			END_IF
		CutterCompleted:
			IF CutterPosition = 0.0 THEN
				CutterDisable := FALSE;
				CutterState := AxisEnabled;
				CutterWorking := FALSE;
			END_IF

			// EMERGENCY STOP
		StopState:
			IF NOT EMERGENCY_STOP AND Cutter.CommandExecuted THEN
				CutterEnable := FALSE;
				CutterDisable := FALSE;
				CutterStopped := TRUE;
				CutterState := Init;
			END_IF

		HaltState:
			IF Cutter.CommandExecuted THEN
				CutterDisable := FALSE;
				CutterEnable := FALSE;
				CutterStopped := TRUE;
				CutterAxisEnable := FALSE;
				CutterState := Init;
			END_IF
	END_CASE

	// Implementing the Homing as in video (as in the first video)
	// Implementing the button (start button, the stop button and the emergency stop)

	// Counter for blink
	Count := Count + 1;
	IF Count = 10 THEN
		ToggleLights := TRUE;
		Count := 0;
	ELSE
		ToggleLights := FALSE;
	END_IF

	// LIGHTS
	IF MachineState = Init THEN
		IF ToggleLights THEN
			GreenLight := NOT GreenLight;
		END_IF
		RedLight := FALSE;
		EmergencyLight := FALSE;

	ELSIF MachineState <> HaltState AND MachineState <> StopState AND MachineState <> CheckReset THEN
		GreenLight := TRUE;
		RedLight := TRUE;
		EmergencyLight := FALSE;
	ELSIF MachineState = StopState OR MachineState = CheckReset THEN
		GreenLight := FALSE;
		RedLight := FALSE;
		IF ToggleLights THEN
			EmergencyLight := NOT EmergencyLight;
		END_IF
	END_IF

	//Conveyor(AxisEnable := ConveyorAxisEnable);
	//ConveyorPosition := Conveyor.ActualPosition;

	//Cutter(AxisEnable := CutterAxisEnable);
	//CutterPosition := Cutter.ActualPosition;

	Conveyor.Axis	:= ADR(gAxis01);
	Conveyor.MpLink	:= ADR(gAxisConveyor);
	RealConveyorSpeed := CONVEYOR_SPEED/10;

	Conveyor.Param.Velocity := INT_TO_REAL(RealConveyorSpeed);
	Conveyor.Param.Acceleration := 100;
	Conveyor.Param.Deceleration := 100;

	Cutter.Axis	:= ADR(gAxis02);
	Cutter.MpLink	:= ADR(gAxisCutter);
	Cutter.MpLinkMaster	:= ADR(gAxisConveyor);

	Cutter.Param.Velocity := CUTTER_SPEED;

	Cutter.Param.Acceleration := 100;
	Cutter.Param.Deceleration := 100;

	CouplingParameters.Cam.LeadIn.CamEnable:= TRUE;
	//CouplingParameters.Cam.MasterStartPosition := 180;

	Cutter.CouplingParam := CouplingParameters;

	Conveyor(AxisEnable := ConveyorAxisEnable);
	ConveyorPosition := Conveyor.ActualPosition;

	Cutter(AxisEnable := CutterAxisEnable);
	CutterPosition := Cutter.ActualPosition;

END_PROGRAM

PROGRAM _EXIT
	(* Insert code here *)

END_PROGRAM
```

#### Variables.var - Local variables
```iecst
(*Conveyor*)
VAR
	Cutter : CamFB;
	Conveyor : CamFB;
	MachineState : State_type;
	ConveyorParameters : MpAxisBasicParType;
END_VAR
(*Cutter*)
VAR
	CutterParameters : MpAxisBasicParType;
END_VAR
(*Coupling*)
VAR
	CouplingParameters : MpAxisCouplingParType;
	ConveyorEnable : BOOL;
	CutterEnable : BOOL;
	InitializeConveyor : BOOL;
	InitializeCutter : BOOL;
	ConveyorDisable : BOOL;
	CutterDisable : BOOL;
	ConveyorState : State_type;
	CutterState : State_type;
	ConveyorAxisEnable : BOOL;
	CutterAxisEnable : BOOL;
	FutureStop : BOOL;
	CoveyorState : BOOL;
	ConveyorStopped : BOOL;
	CutterStopped : BOOL;
	EmergencyStateMachine : INT;
	CamOffset : LREAL;
	CutterWorking : BOOL;
	Count : DINT;
	ToggleLights : BOOL;
END_VAR
```

#### Types.typ - Local data types
```iecst
TYPE
	State_type :
		(
		CutterMoveBackward,
		CutterCompleted,
		ConveyorStopping,
		ConveyorMoving,
		ConveyorStarting,
		AxisEnabled,
		InitializeAxis,
		WaitProduct,
		Initialize,
		Init,
		StopState,
		HaltState,
		WaitForConveyor,
		CheckPower,
		CheckEnable,
		CutterMotion,
		CutterMoveForward,
		ConveyorHolding,
		CutterForward,
		CutterBackward,
		CamEnabled,
		CheckCamUpdate1,
		CheckCamUpdate2,
		CheckReset
		);
END_TYPE
```

### Data object Logical/Cam (Cam)

#### Cam.cam
```
CamProfile (NcSwId=ACP10, MasterAxisVelocity=1, MasterAxisAcceleration=0, DefaultCurveType=Polynomial5, MathematicalNotation=true)
  FixPoint (x=0, IsMathX=true, y=0, IsDefinedDy=false, Dy=0, IsMathDy=true, IsDefinedDdy=false, Ddy=0, IsMathDdy=true, IsDefinedDddy=false, Dddy=0, IsMathDddy=true)
  FixPoint (x=216, IsMathX=true, y=0, IsDefinedDy=false, Dy=0, IsMathDy=true, IsDefinedDdy=false, Ddy=0, IsMathDdy=true, IsDefinedDddy=false, Dddy=0, IsMathDddy=true)
  FixPoint (x=288, IsMathX=true, y=0.5, IsDefinedDy=false, Dy=0, IsMathDy=true, IsDefinedDdy=false, Ddy=0, IsMathDdy=true, IsDefinedDddy=false, Dddy=0, IsMathDddy=true)
  FixPoint (x=360, IsMathX=true, y=0, IsDefinedDy=false, Dy=0, IsMathDy=true, IsDefinedDdy=false, Ddy=0, IsMathDdy=true, IsDefinedDddy=false, Dddy=0, IsMathDddy=true)
  Curve (Type=Polynomial5)
    LeftBoundary (IsDefinedDdy=false, Ddy=0, IsMathDdy=true, IsDefinedDddy=false, Dddy=0, IsMathDddy=true)
    RightBoundary (IsDefinedDdy=false, Ddy=0, IsMathDdy=true, IsDefinedDddy=false, Dddy=0, IsMathDddy=true)
    Spline3 (IsContinuous4Derivative=false, IsDefinedSaddlePoint=false, IsDefinedLineAs2ndSegment=false, IsDefinedSlopeOfLine=false, SlopeOfLine=0, IsMathSlopeOfLine=true)
    Supremum (y=1.7e+308, Dy=1.7e+308, IsMathDy=true, Ddy=1.7e+308, IsMathDdy=true, Dddy=1.7e+308, IsMathDddy=true)
    Infimum (y=-1.7e+308, Dy=-1.7e+308, IsMathDy=true, Ddy=-1.7e+308, IsMathDdy=true, Dddy=-1.7e+308, IsMathDddy=true)
  Curve (Type=Polynomial5)
    LeftBoundary (IsDefinedDdy=false, Ddy=0, IsMathDdy=true, IsDefinedDddy=false, Dddy=0, IsMathDddy=true)
    RightBoundary (IsDefinedDdy=false, Ddy=0, IsMathDdy=true, IsDefinedDddy=false, Dddy=0, IsMathDddy=true)
    Spline3 (IsContinuous4Derivative=false, IsDefinedSaddlePoint=false, IsDefinedLineAs2ndSegment=false, IsDefinedSlopeOfLine=false, SlopeOfLine=0, IsMathSlopeOfLine=true)
    Supremum (y=1.7e+308, Dy=1.7e+308, IsMathDy=true, Ddy=1.7e+308, IsMathDdy=true, Dddy=1.7e+308, IsMathDddy=true)
    Infimum (y=-1.7e+308, Dy=-1.7e+308, IsMathDy=true, Ddy=-1.7e+308, IsMathDdy=true, Dddy=-1.7e+308, IsMathDddy=true)
  Curve (Type=Polynomial5)
    LeftBoundary (IsDefinedDdy=false, Ddy=0, IsMathDdy=true, IsDefinedDddy=false, Dddy=0, IsMathDddy=true)
    RightBoundary (IsDefinedDdy=false, Ddy=0, IsMathDdy=true, IsDefinedDddy=false, Dddy=0, IsMathDddy=true)
    Spline3 (IsContinuous4Derivative=false, IsDefinedSaddlePoint=false, IsDefinedLineAs2ndSegment=false, IsDefinedSlopeOfLine=false, SlopeOfLine=0, IsMathSlopeOfLine=true)
    Supremum (y=1.7e+308, Dy=1.7e+308, IsMathDy=true, Ddy=1.7e+308, IsMathDdy=true, Dddy=1.7e+308, IsMathDddy=true)
    Infimum (y=-1.7e+308, Dy=-1.7e+308, IsMathDy=true, Ddy=-1.7e+308, IsMathDdy=true, Dddy=-1.7e+308, IsMathDddy=true)
  Cam (LeftBoundaryIndex=0, RightBoundaryIndex=3)
    Supremum (y=1.7e+308, Dy=1.7e+308, IsMathDy=true, Ddy=1.7e+308, IsMathDdy=true, Dddy=1.7e+308, IsMathDddy=true)
    Infimum (y=-1.7e+308, Dy=-1.7e+308, IsMathDy=true, Ddy=-1.7e+308, IsMathDdy=true, Dddy=1.7e+308, IsMathDddy=true)
  ChartExtensions
```

### Data object Logical/standstill (Cam)

#### Cam.cam
```
CamProfile (NcSwId=ACP10, MasterAxisVelocity=1, MasterAxisAcceleration=0, DefaultCurveType=Polynomial5, MathematicalNotation=true)
  FixPoint (x=0, IsMathX=true, y=0, IsDefinedDy=false, Dy=0, IsMathDy=true, IsDefinedDdy=false, Ddy=0, IsMathDdy=true, IsDefinedDddy=false, Dddy=0, IsMathDddy=true)
  FixPoint (x=1, IsMathX=true, y=0, IsDefinedDy=false, Dy=0, IsMathDy=true, IsDefinedDdy=false, Ddy=0, IsMathDdy=true, IsDefinedDddy=false, Dddy=0, IsMathDddy=true)
  Curve (Type=Polynomial5)
    LeftBoundary (IsDefinedDdy=false, Ddy=0, IsMathDdy=true, IsDefinedDddy=false, Dddy=0, IsMathDddy=true)
    RightBoundary (IsDefinedDdy=false, Ddy=0, IsMathDdy=true, IsDefinedDddy=false, Dddy=0, IsMathDddy=true)
    Spline3 (IsContinuous4Derivative=false, IsDefinedSaddlePoint=false, IsDefinedLineAs2ndSegment=false, IsDefinedSlopeOfLine=false, SlopeOfLine=0, IsMathSlopeOfLine=true)
    Supremum (y=1.7e+308, Dy=1.7e+308, IsMathDy=true, Ddy=1.7e+308, IsMathDdy=true, Dddy=1.7e+308, IsMathDddy=true)
    Infimum (y=-1.7e+308, Dy=-1.7e+308, IsMathDy=true, Ddy=-1.7e+308, IsMathDdy=true, Dddy=-1.7e+308, IsMathDddy=true)
  Cam (LeftBoundaryIndex=0, RightBoundaryIndex=1)
    Supremum (y=1.7e+308, Dy=1.7e+308, IsMathDy=true, Ddy=1.7e+308, IsMathDdy=true, Dddy=1.7e+308, IsMathDddy=true)
    Infimum (y=-1.7e+308, Dy=-1.7e+308, IsMathDy=true, Ddy=-1.7e+308, IsMathDdy=true, Dddy=1.7e+308, IsMathDddy=true)
  ChartExtensions
```

### Program Logical/PLCopen

#### Types.typ
```iecst
TYPE
	State_type :
		(
		IDLE,
		ENABLE_AXES,
		BELT_MOVING,
		BELT_STOPPING,
		BELT_HOLDING,
		CUTTER_BACK,
		CUTTER_END
		);
END_TYPE
```

#### Main.st
```iecst
PROGRAM _INIT
	(* Insert code here *)

END_PROGRAM

PROGRAM _CYCLIC
	Enable := TRUE;

	IF STOP THEN
		CutterEnable := FALSE;
		ConveyorEnable := FALSE;

		Cutter.AxisCommand := AXIS_STOP;
		Conveyor.AxisCommand := MOVE_ADDITIVE;
		Conveyor.AxisCommand := AXIS_STOP;

		Stop_Light := TRUE;
		Green_Light := FALSE;
		White_Light := FALSE;
		Yellow_Light := FALSE;

		State := IDLE;
	END_IF

	CASE State OF
		IDLE:
			IF START_BUTTON THEN
				CutterEnable := TRUE;
				ConveyorEnable := TRUE;

				Cutter.AxisCommand := AXIS_STOP;
				Conveyor.AxisCommand := AXIS_STOP;

				Stop_Light := FALSE;
				Green_Light := TRUE;
				White_Light := FALSE;
				Yellow_Light := FALSE;

				State := ENABLE_AXES;
			END_IF

		ENABLE_AXES:
			IF Cutter.Status = STANDSTILL AND Conveyor.Status = STANDSTILL THEN
				Conveyor.AxisCommand := MOVE_VELOCITY;

				Stop_Light := FALSE;
				Green_Light := TRUE;
				White_Light := TRUE;
				Yellow_Light := FALSE;

				State := BELT_MOVING;
			END_IF

		BELT_MOVING:
			IF TRIGGER_INPUT THEN
				Conveyor.AxisCommand := MOVE_ADDITIVE;

				State := BELT_STOPPING;
			END_IF

		BELT_STOPPING:
			IF Conveyor.CommandExecuted THEN
				Conveyor.AxisCommand := AXIS_STOP;
				Cutter.AxisCommand := MOVE_ADDITIVE;
				Cutter.Position := CUTTER_END_POSE;

				Stop_Light := FALSE;
				Green_Light := TRUE;
				White_Light := FALSE;
				Yellow_Light := TRUE;

				State := BELT_HOLDING;
			END_IF

		BELT_HOLDING:
			IF Cutter.CommandExecuted THEN
				Cutter.AxisCommand := AXIS_STOP;

				State := CUTTER_BACK;
			END_IF

		CUTTER_BACK:
			IF NOT Cutter.CommandExecuted THEN
				Cutter.AxisCommand := MOVE_ADDITIVE;
				Cutter.Position := -CUTTER_END_POSE;

				State := CUTTER_END;
			END_IF

		CUTTER_END:
			IF Cutter.CommandExecuted THEN
				Cutter.AxisCommand := AXIS_STOP;

				State := ENABLE_AXES;
			END_IF
	END_CASE

	Conveyor.Slave := ADR(gAxis01);
	Conveyor.Position := 2*BELT_DISTANCE;
	Conveyor.Velocity := velocity;
	Conveyor.Acceleration := 100;
	Conveyor.Deceleration := 100;

	Conveyor(AxisEnable := ConveyorEnable);
	ConveyorPosition := Conveyor.ActualPosition;

	Cutter.Slave := ADR(gAxis02);
	Cutter.Velocity := CUTTER_SPEED;
	Cutter.Acceleration := 100;
	Cutter.Deceleration := 100;

	Cutter(AxisEnable := CutterEnable);
	CutterPosition := Cutter.ActualPosition;

END_PROGRAM

PROGRAM _EXIT
	(* Insert code here *)

END_PROGRAM
```

Listed in the project but not available here: Logical/Global.typ, Logical/Libraries/CAMlib/Constants.var, Logical/acp10etxen, Logical/gAxis01obj, Logical/MNG_Global.typ, Logical/InputBridge
